{attribute 'linkalways'} 
{attribute 'no_explicit_call' := 'This FB is a CLASS and must be accessed using methods or properties'}
{attribute 'enable_dynamic_creation'}
FUNCTION_BLOCK _HRESULT EXTENDS AliasDatatypeBase
VAR
	localData : HRESULT;
	activeData : REFERENCE TO HRESULT REF= localData;
	aliasBaseDatatype : _DINT(localData);
END_VAR

PROPERTY PUBLIC Address : PVOID
GET
Address := ADR(activeData);
END_GET
END_PROPERTY

METHOD PUBLIC ClearReference
VAR_INPUT
END_VAR
activeData REF= localData;
SetBaseDatatypeReference();
END_METHOD

METHOD PUBLIC Clone : I_Datatype
VAR
    pClone : POINTER TO _HRESULT;
END_VAR
pClone := __NEW(_HRESULT(InitialValue := Value));
Clone := pClone^;
END_METHOD

METHOD FB_init : BOOL
VAR_INPUT
	bInitRetains : BOOL; // if TRUE, the retain variables are initialized (warm start / cold start)
	bInCopyCode : BOOL;  // if TRUE, the instance afterwards gets moved into the copy code (online change)
	InitialValue : HRESULT;
END_VAR
localData := InitialValue;
SetBaseDatatypeReference();
AddBaseDatatype(aliasBaseDatatype);
END_METHOD

PROPERTY PUBLIC Identifier : T_MAXSTRING
GET
Identifier := 'HRESULT';
END_GET
END_PROPERTY

METHOD PUBLIC MakeReferenceTo
VAR_INPUT
	ReferenceTarget : REFERENCE TO HRESULT;
END_VAR
activeData REF= ReferenceTarget;
SetBaseDatatypeReference();
END_METHOD

METHOD PROTECTED SetBaseDatatypeReference
VAR_INPUT
END_VAR
aliasBaseDatatype.MakeReferenceTo(activeData);
END_METHOD

PROPERTY PUBLIC Size : UDINT
GET
Size := SIZEOF(activeData);
END_GET
END_PROPERTY

METHOD TryMakeReferenceTo : BOOL
VAR_INPUT
	Target : I_Datatype;
END_VAR
VAR
	targetAsAlias : I_AliasDatatype;
	pTargetData : POINTER TO HRESULT;
END_VAR
IF NOT Target.TryResolveAsAliasDatatype(targetAsAlias) THEN
	RETURN;
END_IF

IF targetAsAlias.Identifier <> Identifier THEN
	RETURN;
END_IF

pTargetData := Target.Address;
activeData REF= pTargetData^;
SetBaseDatatypeReference();
TryMakeReferenceTo := TRUE;
END_METHOD

PROPERTY PUBLIC Value : HRESULT
GET
Value := activeData;
END_GET
SET
activeData := Value;
END_SET
END_PROPERTY

END_FUNCTION_BLOCK

(* stored: Version 1.1.0.1, ProductVersion 3.1.4024.12
   POU _HRESULT: Id {9826f510-6a9a-0589-1707-a2f4566837a3}, SpecialFunc None
   Folder Constructor: Id {34c7ada5-c19d-09fc-31cd-1f17e90cc563}
   Folder Protected: Id {cafab655-1853-041b-1823-d2f3fc877384}
   Property Address: Id {353183df-1643-0785-0628-2e3e180ddc80}
   Get Get: Id {6914a22f-266e-02c8-3689-e1f8e5497695}
   Method ClearReference: Id {d5aa871f-b78c-09b6-3f63-b177c3cd8701}
   Method Clone: Id {67b2ac25-bf1c-08b7-2558-1abb64d9be43}
   Method FB_init: Id {7376dfce-ee7c-0dd4-26e9-43c63f7d0b8c}
   Property Identifier: Id {2b4da1fa-fdd1-04c9-217f-f99980bf8f19}
   Get Get: Id {fb672f69-cd14-0da7-3b52-cb4a65be3caf}
   Method MakeReferenceTo: Id {63fc7772-103f-0837-3778-5ec001005eeb}
   Method SetBaseDatatypeReference: Id {7dbd2544-12d4-09b1-360e-b966066bc656}
   Property Size: Id {45fbb52f-934a-0c45-1f67-e6d3b618460b}
   Get Get: Id {8961285f-0244-0d84-21e1-aa542ba07af7}
   Method TryMakeReferenceTo: Id {a4b75e21-0735-0951-21d1-6015acd08bb7}
   Property Value: Id {8c2ed29b-1a32-09bc-0294-a45d826dc13a}
   Get Get: Id {49a8b486-1e1a-0732-04c5-94844c5fd9b4}
   Set Set: Id {0ee3d445-1cdb-04cf-3497-421c1be0161c} *)
